{attribute 'GeneratedUsingTerminal: EK1122-0000-0018'}
{attribute addProperty BoxType "EK1122-0000-0018"}
{attribute addProperty Id "Beckhoff_EL73xxsub_EK1100EK1100_AB5A94672"}
{attribute addProperty CRC "1029908831"}
{attribute addProperty Size "2"}
TYPE Beckhoff_EL73xxEK1122_3D63295F EXTENDS EK1122_AB5A9467 :
STRUCT
	{attribute addProperty Name "Beckhoff_EL73xxsub_EK1100"}
	{attribute addProperty PreviousPort "Beckhoff EL73xxEK1122 : D"}
	Beckhoff_EL73xxsub_EK1100 : EK1100_AB5A9467;
END_STRUCT
END_TYPE

(* stored: Version 1.2.0.0, ProductVersion 3.1.4024.9
   DUT Beckhoff_EL73xxEK1122_3D63295F: Id {db7e25c0-2600-4a41-bf5d-70ca96226889} *)
